Staubli VAL3: insert.pgx

public program insert(string x_sItem, bool& x_bDone)
begin
  // insert a new item
  if isDefined(saveInOut:dOutput[x_sItem])==false
    x_bDone=true
    insert(saveInOut:dOutput[x_sItem])
  else
    // already exist
    x_bDone=false
  endIf

end
